FUNCTION_BLOCK FB_PID
VAR_INPUT
	xSet:	REAL; 	// Set value
	xAct:	REAL;	// measured Value	

	Kp  :  	REAL;  	// proportional factor
	Ti  :  	REAL;  	// integral time
	Td  :	REAL; 	// derivative time
		
	LimLow	:	REAL; 	// lower limit of output
	LimHigh	: 	REAL; 	// upper limit of output
	StartY	:	REAL;	// Y to use as offset
	
	bReverseActing 	:	BOOL;	// True for reverse acting
	
	RST		:	BOOL; 	// Reset
END_VAR
VAR_OUTPUT
	Y : REAL;		// controller output
	LIM : BOOL;		// True, if output reaches LimLow or LimHigh
END_VAR
VAR
	e			:  REAL;		// control difference
	yOffset		:  REAL	:= 0;		// constant offset used on Y	
	fbDerivative :  FT_DERIV; 	// function block for derivation
	fbIntegrate  :	FB_Integrate;	// function block for integration
END_VAR

IF StartY <> 0 THEN
	yOffset := StartY;
	IF RST THEN
		fbIntegrate(RST:=TRUE, inStart:=0);
	END_IF
END_IF

//determine direct or reverse acting
IF bReverseActing THEN
	e := xAct - xSet;
ELSE
	e := xSet - xAct;	
END_IF;

IF Ti>0 THEN
	//derivative and integral calculation
	fbDerivative(in:=e,run:=TRUE);
	fbIntegrate(run:= TRUE, in := e, RST:=RST);
	Y := Kp * (e + 1/Ti * fbIntegrate.out + Td * fbDerivative.out) + yOffset;
ELSE
	//derivative  calculation
	fbDerivative(in:=e,run:=TRUE);
	Y := Kp * (e + Td * fbDerivative.out) + yOffset;
END_IF

//Check limits and Anti-wind up
IF Y < LimLow AND NOT RST THEN
	Y := LimLow;
	LIM := TRUE;
	fbIntegrate(RST:=TRUE, inStart:=(Y/Kp - e)*Ti);
ELSIF Y > LimHigh AND NOT RST THEN
	Y := LimHigh;
	LIM := TRUE;
	fbIntegrate(RST:=TRUE, inStart:=(Y/Kp - e)*Ti);
ELSE
	LIM := FALSE;	
END_IF

(*
pos 23.10.2020:
- no anti-wind up on reset
- possibility to provide an offset value for Y

aku 24.09.2019: first implementation
*)

END_FUNCTION_BLOCK

(* stored: Version 1.1.0.1, ProductVersion 3.1.4024.3
   POU FB_PID: Id {9148ddd9-4f6e-4c4f-98a6-9a43459fe84e}, SpecialFunc None *)
